# EPICS substitutions: HidenRGAApp/Db/asynRecord.substitutions
file asynRecord.template
{
	pattern	{ P		, R		, PORT		, ADDR	, OMAX	, IMAX	}
		{ XF:03-VA	, "{RGAC:1}"	, XF03VA_RGAC1	, 0	, 0	, 0	}
}
